Universal Robots PolyScope program: phoneBoxing.urp

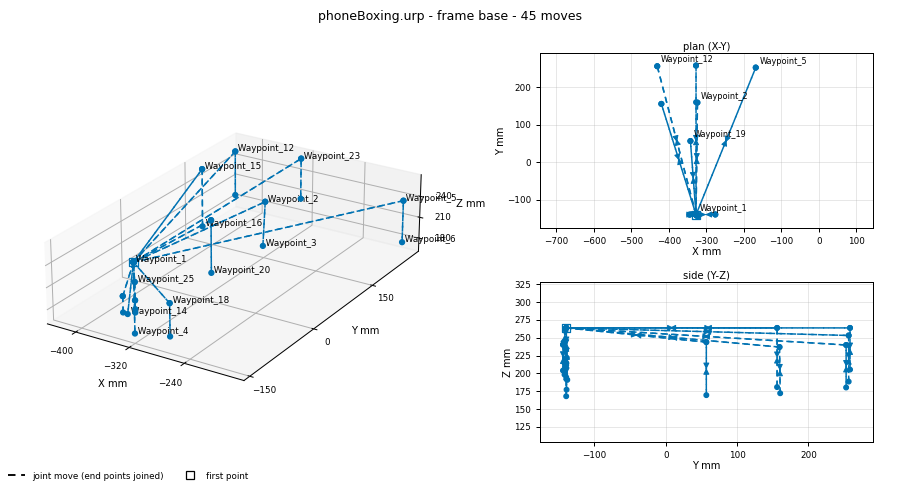
[picture p0: tool path of phoneBoxing.urp in frame base, 45 of 45 moves have a stored position in this frame; points joined in program order, loops and branches not executed]
Program phoneBoxing (installation=schmalz directory=/programs createdIn=5.2.0.61336 lastSavedIn=5.2.0.61336 robotSerialNumber=20185300040)
Calibrated DH parameters: a=[-0.000128, -0.221415, -0.194849, 0.000098, -0.000148, 0]; d=[0.152137, 33.879231, 13.968137, -47.716378, 0.085395, 0.092257]; alpha=[1.57105, 0.003021, -0.001826, 1.571145, -1.57192, 0]; deltaTheta=[0, 0.433042, -0.854582, 0.421536, 0.000002, 0]
Robot Program (runOnlyOnce=false)
  Set DigitalOutput pin=tool_out[0]; digitalValue=1
  MoveJ speed 60 deg/s, acceleration 80 deg/s^2 (useActiveTCP=true) feature=Base
    Waypoint Waypoint_1: TCP in base x=-327.452 y=-139.556 z=263.707 mm, rx=-1.7751 ry=-2.5819 rz=0.0078 rad; joints [1.569, -81.889, 92.27, -101, -90.042, -19.554] deg
    Waypoint Waypoint_2: TCP in base x=-323.67 y=159.433 z=236.886 mm, rx=-1.7751 ry=-2.5818 rz=0.0079 rad; joints [-47.55, -79.212, 96.426, -107.682, -89.596, -68.674] deg
    Waypoint Waypoint_3: TCP in base x=-327.514 y=160.36 z=172.126 mm, rx=-1.7751 ry=-2.5818 rz=0.0079 rad; joints [-47.165, -71.608, 105.724, -124.589, -89.583, -68.307] deg
  Set DigitalOutput pin=tool_out[0]; digitalValue=0
  Set DigitalOutput pin=tool_out[1]; digitalValue=1
  Wait Sleep waitTime=0.3
  MoveJ speed 60 deg/s, acceleration 80 deg/s^2 (useActiveTCP=true) feature=Base
    Waypoint Waypoint_2: TCP in base x=-323.67 y=159.433 z=236.886 mm, rx=-1.7751 ry=-2.5818 rz=0.0079 rad; joints [-47.55, -79.212, 96.426, -107.682, -89.596, -68.674] deg
    Waypoint Waypoint_1: TCP in base x=-327.452 y=-139.556 z=263.707 mm, rx=-1.7751 ry=-2.5819 rz=0.0078 rad; joints [1.569, -81.889, 92.27, -101, -90.042, -19.554] deg
    Waypoint Waypoint_4: TCP in base x=-327.453 y=-139.54 z=167.939 mm, rx=-1.7752 ry=-2.5818 rz=0.0078 rad; joints [1.586, -72.861, 108.957, -126.716, -90.022, -19.561] deg
  Set DigitalOutput pin=tool_out[1]; digitalValue=0
  Set DigitalOutput pin=tool_out[0]; digitalValue=1
  Wait Sleep waitTime=0.3
  MoveJ speed 60 deg/s, acceleration 80 deg/s^2 (useActiveTCP=true) feature=Base
    Waypoint Waypoint_1: TCP in base x=-327.452 y=-139.556 z=263.707 mm, rx=-1.7751 ry=-2.5819 rz=0.0078 rad; joints [1.569, -81.889, 92.27, -101, -90.042, -19.554] deg
    Waypoint Waypoint_12: TCP in base x=-430.92 y=256.357 z=253.104 mm, rx=-1.7751 ry=-2.5819 rz=0.0078 rad; joints [-46.007, -39.892, 30.083, -80.668, -89.53, -66.993] deg
    Waypoint Waypoint_13: TCP in base x=-430.922 y=256.355 z=188.454 mm, rx=-1.7751 ry=-2.582 rz=0.0079 rad; joints [-45.976, -40.277, 48.231, -98.425, -89.543, -66.993] deg
  Set DigitalOutput pin=tool_out[0]; digitalValue=0
  Set DigitalOutput pin=tool_out[1]; digitalValue=1
  Wait Sleep waitTime=0.3
  MoveJ speed 60 deg/s, acceleration 80 deg/s^2 (useActiveTCP=true) feature=Base
    Waypoint Waypoint_12: TCP in base x=-430.92 y=256.357 z=253.104 mm, rx=-1.7751 ry=-2.5819 rz=0.0078 rad; joints [-46.007, -39.892, 30.083, -80.668, -89.53, -66.993] deg
    Waypoint Waypoint_1: TCP in base x=-327.452 y=-139.556 z=263.707 mm, rx=-1.7751 ry=-2.5819 rz=0.0078 rad; joints [1.569, -81.889, 92.27, -101, -90.042, -19.554] deg
    Waypoint Waypoint_14: TCP in base x=-338.713 y=-138.003 z=190.891 mm, rx=-1.7752 ry=-2.5819 rz=0.0078 rad; joints [1.27, -73.715, 102.831, -119.733, -90.022, -19.87] deg
  Set DigitalOutput pin=tool_out[1]; digitalValue=0
  Set DigitalOutput pin=tool_out[0]; digitalValue=1
  Wait Sleep waitTime=0.3
  MoveJ speed 60 deg/s, acceleration 80 deg/s^2 (useActiveTCP=true) feature=Base
    Waypoint Waypoint_1: TCP in base x=-327.452 y=-139.556 z=263.707 mm, rx=-1.7751 ry=-2.5819 rz=0.0078 rad; joints [1.569, -81.889, 92.27, -101, -90.042, -19.554] deg
    Waypoint Waypoint_15: TCP in base x=-419.971 y=156 z=263.701 mm, rx=-1.7751 ry=-2.5819 rz=0.0078 rad; joints [-37.44, -58.239, 59.346, -91.632, -89.626, -58.493] deg
    Waypoint Waypoint_16: TCP in base x=-419.974 y=155.991 z=180.751 mm, rx=-1.7752 ry=-2.5819 rz=0.0078 rad; joints [-37.413, -54.145, 75.391, -111.769, -89.628, -58.491] deg
  Set DigitalOutput pin=tool_out[0]; digitalValue=0
  Set DigitalOutput pin=tool_out[1]; digitalValue=1
  Wait Sleep waitTime=0.3
  MoveJ speed 60 deg/s, acceleration 80 deg/s^2 (useActiveTCP=true) feature=Base
    Waypoint Waypoint_15: TCP in base x=-419.971 y=156 z=263.701 mm, rx=-1.7751 ry=-2.5819 rz=0.0078 rad; joints [-37.44, -58.239, 59.346, -91.632, -89.626, -58.493] deg
    Waypoint Waypoint_1: TCP in base x=-327.452 y=-139.556 z=263.707 mm, rx=-1.7751 ry=-2.5819 rz=0.0078 rad; joints [1.569, -81.889, 92.27, -101, -90.042, -19.554] deg
    Waypoint Waypoint_18: TCP in base x=-276.046 y=-139.027 z=221.813 mm, rx=-1.7751 ry=-2.5819 rz=0.0078 rad; joints [1.773, -90.791, 113.62, -113.448, -90.072, -19.386] deg
    Waypoint Waypoint_17: TCP in base x=-276.041 y=-139.034 z=177.152 mm, rx=-1.7751 ry=-2.5819 rz=0.0078 rad; joints [1.781, -84.963, 121.306, -126.961, -90.052, -19.394] deg
  Set DigitalOutput pin=tool_out[1]; digitalValue=0
  Set DigitalOutput pin=tool_out[0]; digitalValue=1
  Wait Sleep waitTime=0.3
  MoveJ speed 60 deg/s, acceleration 80 deg/s^2 (useActiveTCP=true) feature=Base
    Waypoint Waypoint_18: TCP in base x=-276.046 y=-139.027 z=221.813 mm, rx=-1.7751 ry=-2.5819 rz=0.0078 rad; joints [1.773, -90.791, 113.62, -113.448, -90.072, -19.386] deg
    Waypoint Waypoint_1: TCP in base x=-327.452 y=-139.556 z=263.707 mm, rx=-1.7751 ry=-2.5819 rz=0.0078 rad; joints [1.569, -81.889, 92.27, -101, -90.042, -19.554] deg
    Waypoint Waypoint_19: TCP in base x=-342.382 y=56.848 z=243.737 mm, rx=-1.7751 ry=-2.5819 rz=0.0078 rad; joints [-31.601, -83.04, 99.081, -106.595, -89.737, -52.734] deg
    Waypoint Waypoint_20: TCP in base x=-342.381 y=56.835 z=169.465 mm, rx=-1.775 ry=-2.5819 rz=0.0078 rad; joints [-31.586, -75.052, 111.469, -126.973, -89.715, -52.744] deg
  Set DigitalOutput pin=tool_out[0]; digitalValue=0
  Set DigitalOutput pin=tool_out[1]; digitalValue=1
  Wait Sleep waitTime=0.3
  MoveJ speed 60 deg/s, acceleration 80 deg/s^2 (useActiveTCP=true) feature=Base
    Waypoint Waypoint_19: TCP in base x=-342.382 y=56.848 z=243.737 mm, rx=-1.7751 ry=-2.5819 rz=0.0078 rad; joints [-31.601, -83.04, 99.081, -106.595, -89.737, -52.734] deg
    Waypoint Waypoint_1: TCP in base x=-327.452 y=-139.556 z=263.707 mm, rx=-1.7751 ry=-2.5819 rz=0.0078 rad; joints [1.569, -81.889, 92.27, -101, -90.042, -19.554] deg
    Waypoint Waypoint_21: TCP in base x=-344.452 y=-139.434 z=214.216 mm, rx=-1.775 ry=-2.5819 rz=0.0078 rad; joints [1.48, -74.792, 97.326, -113.154, -90.027, -19.655] deg
    Waypoint Waypoint_22: TCP in base x=-344.462 y=-139.416 z=192.14 mm, rx=-1.7751 ry=-2.5818 rz=0.0078 rad; joints [1.481, -72.54, 100.831, -118.912, -90.023, -19.655] deg
  Set DigitalOutput pin=tool_out[1]; digitalValue=0
  Set DigitalOutput pin=tool_out[0]; digitalValue=1
  Wait Sleep waitTime=0.3
  MoveJ speed 60 deg/s, acceleration 80 deg/s^2 (useActiveTCP=true) feature=Base
    Waypoint Waypoint_21: TCP in base x=-344.452 y=-139.434 z=214.216 mm, rx=-1.775 ry=-2.5819 rz=0.0078 rad; joints [1.48, -74.792, 97.326, -113.154, -90.027, -19.655] deg
    Waypoint Waypoint_1: TCP in base x=-327.452 y=-139.556 z=263.707 mm, rx=-1.7751 ry=-2.5819 rz=0.0078 rad; joints [1.569, -81.889, 92.27, -101, -90.042, -19.554] deg
    Waypoint Waypoint_5: TCP in base x=-168.177 y=252.767 z=239.743 mm, rx=-1.7751 ry=-2.5819 rz=0.0078 rad; joints [-82.008, -93.796, 111.17, -107.548, -89.481, -103.158] deg
    Waypoint Waypoint_6: TCP in base x=-168.176 y=252.766 z=180.191 mm, rx=-1.7751 ry=-2.5819 rz=0.0079 rad; joints [-81.999, -86.859, 122.171, -125.485, -89.461, -103.172] deg
  Set DigitalOutput pin=tool_out[0]; digitalValue=0
  Set DigitalOutput pin=tool_out[1]; digitalValue=1
  Wait Sleep waitTime=0.3
  MoveJ speed 60 deg/s, acceleration 80 deg/s^2 (useActiveTCP=true) feature=Base
    Waypoint Waypoint_5: TCP in base x=-168.177 y=252.767 z=239.743 mm, rx=-1.7751 ry=-2.5819 rz=0.0078 rad; joints [-82.008, -93.796, 111.17, -107.548, -89.481, -103.158] deg
    Waypoint Waypoint_1: TCP in base x=-327.452 y=-139.556 z=263.707 mm, rx=-1.7751 ry=-2.5819 rz=0.0078 rad; joints [1.569, -81.889, 92.27, -101, -90.042, -19.554] deg
    Waypoint Waypoint_7: TCP in base x=-324.75 y=-141.69 z=214.379 mm, rx=-1.7751 ry=-2.5819 rz=0.0078 rad; joints [1.967, -78.872, 102.518, -114.265, -90.041, -19.173] deg
    Waypoint Waypoint_8: TCP in base x=-324.729 y=-141.718 z=198.019 mm, rx=-1.775 ry=-2.582 rz=0.0078 rad; joints [1.975, -77.149, 105.216, -118.682, -90.035, -19.175] deg
  Set DigitalOutput pin=tool_out[1]; digitalValue=0
  Set DigitalOutput pin=tool_out[0]; digitalValue=1
  Wait Sleep waitTime=0.3
  MoveJ speed 60 deg/s, acceleration 80 deg/s^2 (useActiveTCP=true) feature=Base
    Waypoint Waypoint_7: TCP in base x=-324.75 y=-141.69 z=214.379 mm, rx=-1.7751 ry=-2.5819 rz=0.0078 rad; joints [1.967, -78.872, 102.518, -114.265, -90.041, -19.173] deg
    Waypoint Waypoint_1: TCP in base x=-327.452 y=-139.556 z=263.707 mm, rx=-1.7751 ry=-2.5819 rz=0.0078 rad; joints [1.569, -81.889, 92.27, -101, -90.042, -19.554] deg
    Waypoint Waypoint_23: TCP in base x=-327.461 y=258.235 z=263.71 mm, rx=-1.7751 ry=-2.5819 rz=0.0078 rad; joints [-56.642, -66.584, 72.07, -95.885, -89.51, -77.724] deg
    Waypoint Waypoint_24: TCP in base x=-327.455 y=258.245 z=205.291 mm, rx=-1.7751 ry=-2.5819 rz=0.0079 rad; joints [-56.626, -63.48, 83.54, -110.456, -89.508, -77.726] deg
  Set DigitalOutput pin=tool_out[0]; digitalValue=0
  Set DigitalOutput pin=tool_out[1]; digitalValue=1
  MoveJ speed 60 deg/s, acceleration 80 deg/s^2 (useActiveTCP=true) feature=Base
    Waypoint Waypoint_23: TCP in base x=-327.461 y=258.235 z=263.71 mm, rx=-1.7751 ry=-2.5819 rz=0.0078 rad; joints [-56.642, -66.584, 72.07, -95.885, -89.51, -77.724] deg
    Waypoint Waypoint_1: TCP in base x=-327.452 y=-139.556 z=263.707 mm, rx=-1.7751 ry=-2.5819 rz=0.0078 rad; joints [1.569, -81.889, 92.27, -101, -90.042, -19.554] deg
    Waypoint Waypoint_25: TCP in base x=-323.041 y=-144.068 z=240.247 mm, rx=-1.7752 ry=-2.582 rz=0.0079 rad; joints [2.387, -81.145, 97.873, -107.344, -90.046, -18.745] deg
    Waypoint Waypoint_26: TCP in base x=-323.04 y=-144.064 z=203.937 mm, rx=-1.7752 ry=-2.582 rz=0.0078 rad; joints [2.394, -77.946, 104.447, -117.114, -90.04, -18.748] deg
  Set DigitalOutput pin=tool_out[1]; digitalValue=0
  Set DigitalOutput pin=tool_out[0]; digitalValue=1
  Wait Sleep waitTime=0.3
  MoveJ speed 60 deg/s, acceleration 80 deg/s^2 (useActiveTCP=true) feature=Base
    Waypoint Waypoint_25: TCP in base x=-323.041 y=-144.068 z=240.247 mm, rx=-1.7752 ry=-2.582 rz=0.0079 rad; joints [2.387, -81.145, 97.873, -107.344, -90.046, -18.745] deg
    Waypoint Waypoint_1: TCP in base x=-327.452 y=-139.556 z=263.707 mm, rx=-1.7751 ry=-2.5819 rz=0.0078 rad; joints [1.569, -81.889, 92.27, -101, -90.042, -19.554] deg
  Halt
